// TIA Portal V16 export
// export: Created 2021-03-13T12:01:04.9234084Z, ExportSetting WithDefaults, DisplayName Totally Integrated Automation Portal, DisplayVersion V16 Update 3, DisplayName TIA Portal Version Control Interface, DisplayVersion V16 Update 2, DisplayName TIA Portal Openness, DisplayVersion V16 Update 3, DisplayName STEP 7 Professional, DisplayVersion V16 Update 3, DisplayName STEP 7 Safety, DisplayVersion V16, DisplayName WinCC Professional, DisplayVersion V16 Update 3
TYPE "UT01001_St_SysLicence"
TITLE = Static UDT — Sys - Licence Information
// Licence Information
// stored: IsFailsafeCompliant false
   STRUCT
      LICENCE_TYPE { ExternalWritable := 'False'} : String[20];   // Licence information — type of licence
      COPYRIGHT { ExternalWritable := 'False'} : String[30];   // Licence information — copyright (year and name)
   END_STRUCT;
END_TYPE
